# EPICS StreamDevice protocol: SPINFLIPPER306015/SPINFLIPPER-IOC-01App/protocol/SPINFLIPPER.proto
#InTerminator = ';';
#OutTerminator = '*';
ReplyTimeout = 2000;

readGuideTemp {
    out "TGUI";
    in "%f";
    ExtraInput = Ignore;
}

readMaxGuideTemp {
    out "GLIM";
    in "%f";
    ExtraInput = Ignore;
}

readFlipState {
    out "FLIP";
    in "%{OFF|ON}";
    ExtraInput = Ignore;
}

readCoilTemp {
    out "TCOI";
    in "%f";
    ExtraInput = Ignore;
}

readMaxCoilTemp {
    out "CLIM";
    in "%f";
    ExtraInput = Ignore;
}

readFlipCurrentSetpoint {
    out "SETI";
    in "%f";
    ExtraInput = Ignore;
}

readFlipCurrent {
    out "IRMS";
    in "%f";
    ExtraInput = Ignore;
}

readFlipFreq {
    out "FREQ";
    in "%f";
    ExtraInput = Ignore;
}

readAlarmState {
    out "ALRM";
    in "%s";
    ExtraInput = Ignore;
}

readMode {
    out "MODE";
    in "%s";
    ExtraInput = Ignore;
}

writeMaxCoilTemp {
    out "LIMC %f";
    in "#";
    ExtraInput = Ignore;
}

writeMaxGuideTemp {
    out "LIMG %f";
    in "#";
    ExtraInput = Ignore;
}

writeRmsFlipCurrent {
    out "ISET %f";
    in "#";
    ExtraInput = Ignore;
}

toggleFlipState {
    out "FL%{OF|ON}";
    in "%{-|~}";
    ExtraInput = Ignore;
}

reset {
    out "RSET";
    in "READY";
    ExtraInput = Ignore;
}
